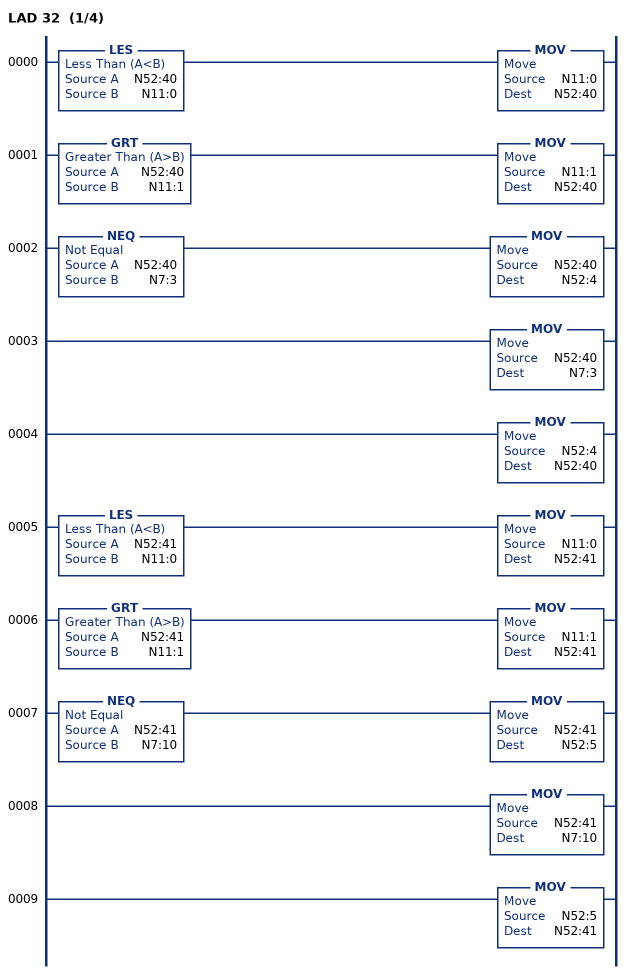
% Rung: 0 %
SOR LES N52:40 N11:0 MOV N11:0 N52:40 EOR
% Rung: 1 %
SOR GRT N52:40 N11:1 MOV N11:1 N52:40 EOR
% Rung: 2 %
SOR NEQ N52:40 N7:3 MOV N52:40 N52:4 EOR
% Rung: 3 %
SOR MOV N52:40 N7:3 EOR
% Rung: 4 %
SOR MOV N52:4 N52:40 EOR
% Rung: 5 %
SOR LES N52:41 N11:0 MOV N11:0 N52:41 EOR
% Rung: 6 %
SOR GRT N52:41 N11:1 MOV N11:1 N52:41 EOR
% Rung: 7 %
SOR NEQ N52:41 N7:10 MOV N52:41 N52:5 EOR
% Rung: 8 %
SOR MOV N52:41 N7:10 EOR
% Rung: 9 %
SOR MOV N52:5 N52:41 EOR

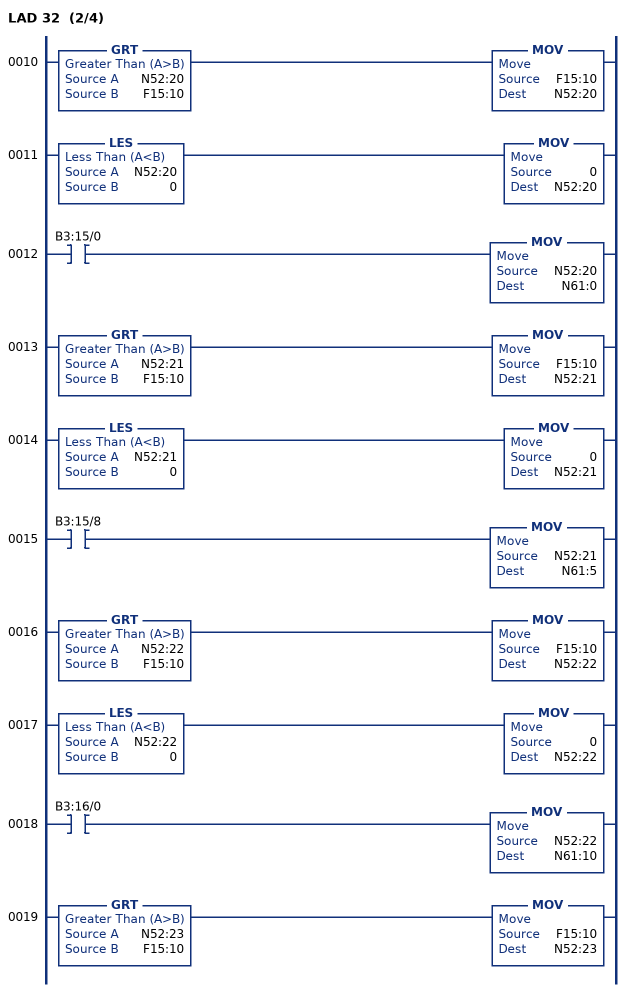
% Rung: 10 %
SOR GRT N52:20 F15:10 MOV F15:10 N52:20 EOR
% Rung: 11 %
SOR LES N52:20 0 MOV 0 N52:20 EOR
% Rung: 12 %
SOR XIC B3:15/0 MOV N52:20 N61:0 EOR
% Rung: 13 %
SOR GRT N52:21 F15:10 MOV F15:10 N52:21 EOR
% Rung: 14 %
SOR LES N52:21 0 MOV 0 N52:21 EOR
% Rung: 15 %
SOR XIC B3:15/8 MOV N52:21 N61:5 EOR
% Rung: 16 %
SOR GRT N52:22 F15:10 MOV F15:10 N52:22 EOR
% Rung: 17 %
SOR LES N52:22 0 MOV 0 N52:22 EOR
% Rung: 18 %
SOR XIC B3:16/0 MOV N52:22 N61:10 EOR
% Rung: 19 %
SOR GRT N52:23 F15:10 MOV F15:10 N52:23 EOR

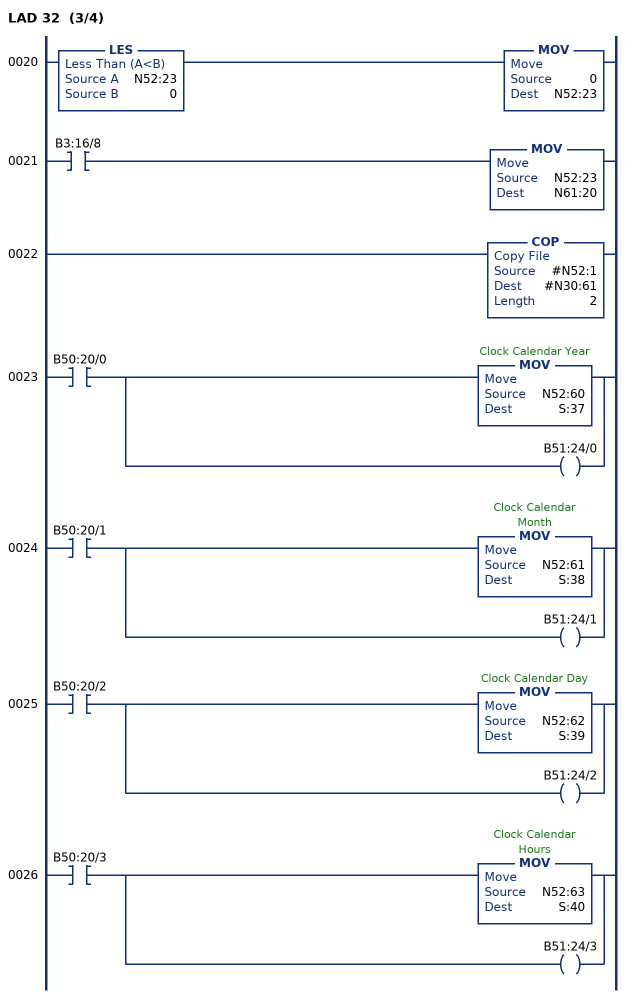
% Rung: 20 %
SOR LES N52:23 0 MOV 0 N52:23 EOR
% Rung: 21 %
SOR XIC B3:16/8 MOV N52:23 N61:20 EOR
% Rung: 22 %
SOR COP #N52:1 #N30:61 2 EOR
% Rung: 23 %
SOR XIC B50:20/0 BST MOV N52:60 S:37 NXB OTE B51:24/0 BND EOR
%   S:37  "Clock Calendar Year" %
% Rung: 24 %
SOR XIC B50:20/1 BST MOV N52:61 S:38 NXB OTE B51:24/1 BND EOR
%   S:38  "Clock Calendar Month" %
% Rung: 25 %
SOR XIC B50:20/2 BST MOV N52:62 S:39 NXB OTE B51:24/2 BND EOR
%   S:39  "Clock Calendar Day" %
% Rung: 26 %
SOR XIC B50:20/3 BST MOV N52:63 S:40 NXB OTE B51:24/3 BND EOR
%   S:40  "Clock Calendar Hours" %

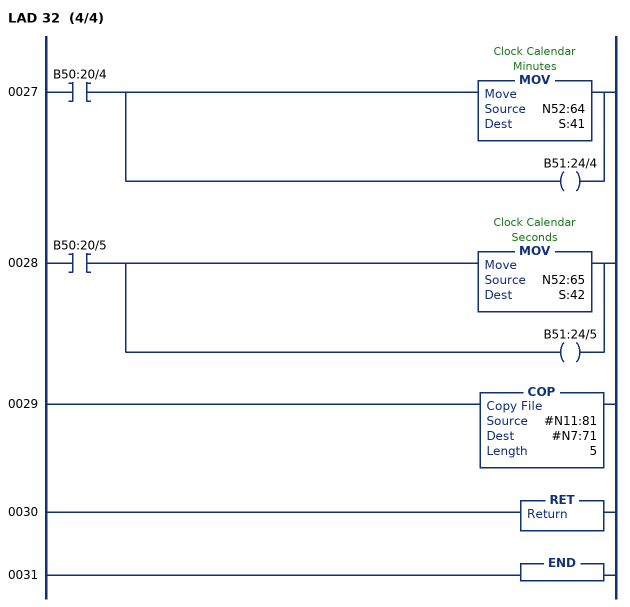
% Rung: 27 %
SOR XIC B50:20/4 BST MOV N52:64 S:41 NXB OTE B51:24/4 BND EOR
%   S:41  "Clock Calendar Minutes" %
% Rung: 28 %
SOR XIC B50:20/5 BST MOV N52:65 S:42 NXB OTE B51:24/5 BND EOR
%   S:42  "Clock Calendar Seconds" %
% Rung: 29 %
SOR COP #N11:81 #N7:71 5 EOR
% Rung: 30 %
SOR RET EOR
% Rung: 31 %
SOR END EOR

LADDER 33
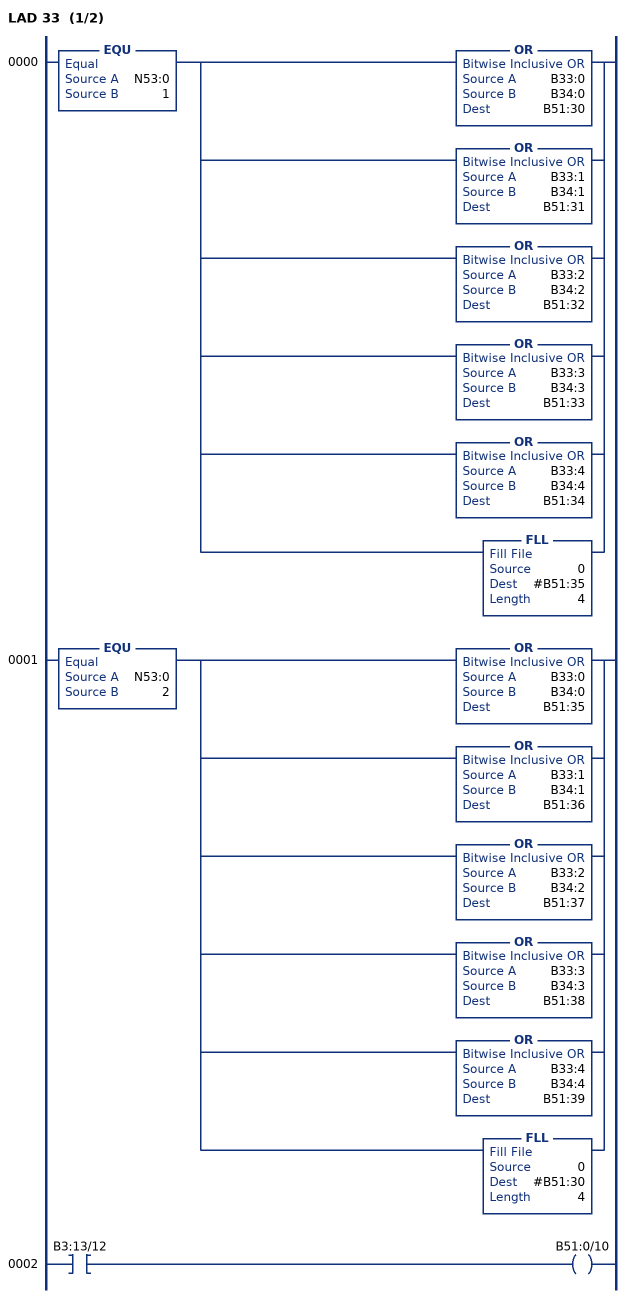
% Rung: 0 %
SOR EQU N53:0 1 BST OR B33:0 B34:0 B51:30 NXB OR B33:1 B34:1 B51:31 NXB OR B33:2 B34:2 B51:32 NXB OR B33:3 B34:3 B51:33 NXB OR B33:4 B34:4 B51:34 NXB FLL 0 #B51:35 4 BND EOR
% Rung: 1 %
SOR EQU N53:0 2 BST OR B33:0 B34:0 B51:35 NXB OR B33:1 B34:1 B51:36 NXB OR B33:2 B34:2 B51:37 NXB OR B33:3 B34:3 B51:38 NXB OR B33:4 B34:4 B51:39 NXB FLL 0 #B51:30 4 BND EOR
% Rung: 2 %
SOR XIC B3:13/12 OTE B51:0/10 EOR

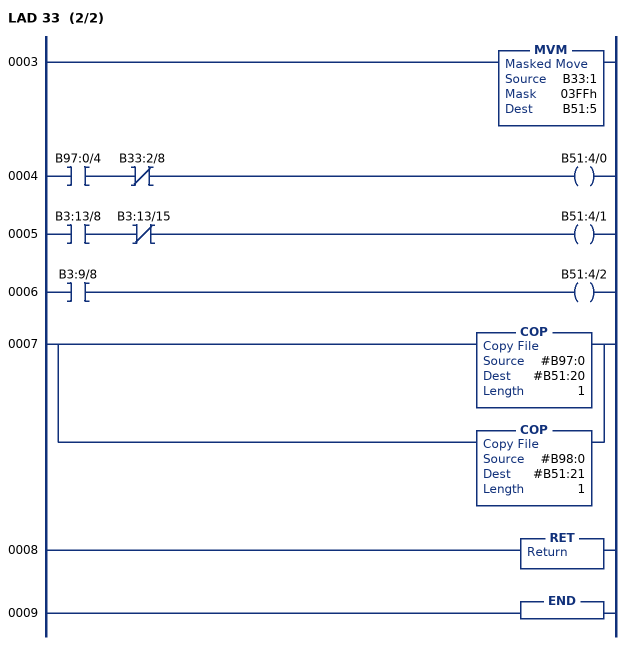
% Rung: 3 %
SOR MVM B33:1 03FFh B51:5 EOR
% Rung: 4 %
SOR XIC B97:0/4 XIO B33:2/8 OTE B51:4/0 EOR
% Rung: 5 %
SOR XIC B3:13/8 XIO B3:13/15 OTE B51:4/1 EOR
% Rung: 6 %
SOR XIC B3:9/8 OTE B51:4/2 EOR
% Rung: 7 %
SOR BST COP #B97:0 #B51:20 1 NXB COP #B98:0 #B51:21 1 BND EOR
% Rung: 8 %
SOR RET EOR
% Rung: 9 %
SOR END EOR

LADDER 34
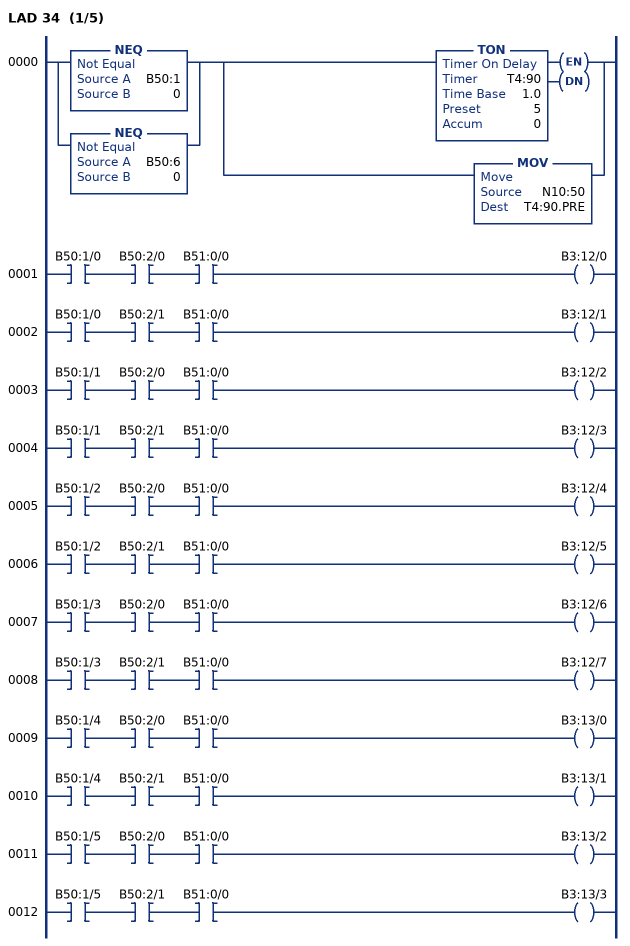
% Rung: 0 %
SOR BST NEQ B50:1 0 NXB NEQ B50:6 0 BND BST TON T4:90 1.0 5 0 NXB MOV N10:50 T4:90.PRE BND EOR
% Rung: 1 %
SOR XIC B50:1/0 XIC B50:2/0 XIC B51:0/0 OTE B3:12/0 EOR
% Rung: 2 %
SOR XIC B50:1/0 XIC B50:2/1 XIC B51:0/0 OTE B3:12/1 EOR
% Rung: 3 %
SOR XIC B50:1/1 XIC B50:2/0 XIC B51:0/0 OTE B3:12/2 EOR
% Rung: 4 %
SOR XIC B50:1/1 XIC B50:2/1 XIC B51:0/0 OTE B3:12/3 EOR
% Rung: 5 %
SOR XIC B50:1/2 XIC B50:2/0 XIC B51:0/0 OTE B3:12/4 EOR
% Rung: 6 %
SOR XIC B50:1/2 XIC B50:2/1 XIC B51:0/0 OTE B3:12/5 EOR
% Rung: 7 %
SOR XIC B50:1/3 XIC B50:2/0 XIC B51:0/0 OTE B3:12/6 EOR
% Rung: 8 %
SOR XIC B50:1/3 XIC B50:2/1 XIC B51:0/0 OTE B3:12/7 EOR
% Rung: 9 %
SOR XIC B50:1/4 XIC B50:2/0 XIC B51:0/0 OTE B3:13/0 EOR
% Rung: 10 %
SOR XIC B50:1/4 XIC B50:2/1 XIC B51:0/0 OTE B3:13/1 EOR
% Rung: 11 %
SOR XIC B50:1/5 XIC B50:2/0 XIC B51:0/0 OTE B3:13/2 EOR
% Rung: 12 %
SOR XIC B50:1/5 XIC B50:2/1 XIC B51:0/0 OTE B3:13/3 EOR

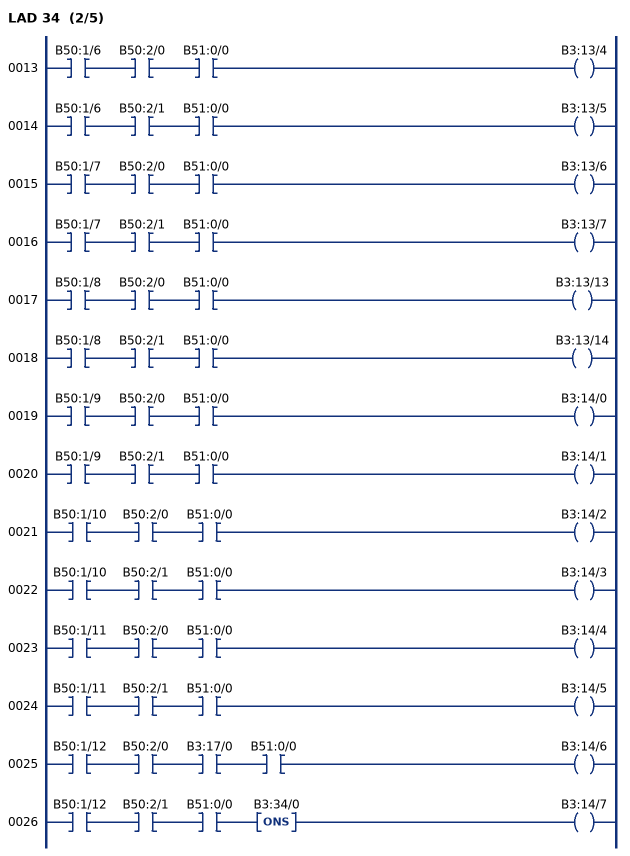
% Rung: 13 %
SOR XIC B50:1/6 XIC B50:2/0 XIC B51:0/0 OTE B3:13/4 EOR
% Rung: 14 %
SOR XIC B50:1/6 XIC B50:2/1 XIC B51:0/0 OTE B3:13/5 EOR
% Rung: 15 %
SOR XIC B50:1/7 XIC B50:2/0 XIC B51:0/0 OTE B3:13/6 EOR
% Rung: 16 %
SOR XIC B50:1/7 XIC B50:2/1 XIC B51:0/0 OTE B3:13/7 EOR
% Rung: 17 %
SOR XIC B50:1/8 XIC B50:2/0 XIC B51:0/0 OTE B3:13/13 EOR
% Rung: 18 %
SOR XIC B50:1/8 XIC B50:2/1 XIC B51:0/0 OTE B3:13/14 EOR
% Rung: 19 %
SOR XIC B50:1/9 XIC B50:2/0 XIC B51:0/0 OTE B3:14/0 EOR
% Rung: 20 %
SOR XIC B50:1/9 XIC B50:2/1 XIC B51:0/0 OTE B3:14/1 EOR
% Rung: 21 %
SOR XIC B50:1/10 XIC B50:2/0 XIC B51:0/0 OTE B3:14/2 EOR
% Rung: 22 %
SOR XIC B50:1/10 XIC B50:2/1 XIC B51:0/0 OTE B3:14/3 EOR
% Rung: 23 %
SOR XIC B50:1/11 XIC B50:2/0 XIC B51:0/0 OTE B3:14/4 EOR
% Rung: 24 %
SOR XIC B50:1/11 XIC B50:2/1 XIC B51:0/0 OTE B3:14/5 EOR
% Rung: 25 %
SOR XIC B50:1/12 XIC B50:2/0 XIC B3:17/0 XIC B51:0/0 OTE B3:14/6 EOR
% Rung: 26 %
SOR XIC B50:1/12 XIC B50:2/1 XIC B51:0/0 OSR B3:34/0 OTE B3:14/7 EOR

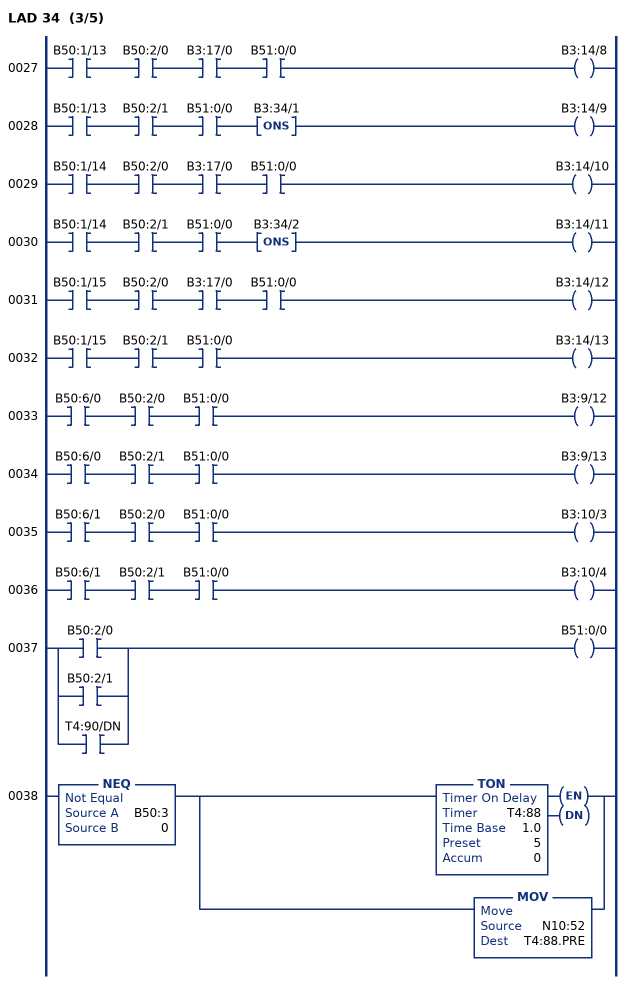
% Rung: 27 %
SOR XIC B50:1/13 XIC B50:2/0 XIC B3:17/0 XIC B51:0/0 OTE B3:14/8 EOR
% Rung: 28 %
SOR XIC B50:1/13 XIC B50:2/1 XIC B51:0/0 OSR B3:34/1 OTE B3:14/9 EOR
% Rung: 29 %
SOR XIC B50:1/14 XIC B50:2/0 XIC B3:17/0 XIC B51:0/0 OTE B3:14/10 EOR
% Rung: 30 %
SOR XIC B50:1/14 XIC B50:2/1 XIC B51:0/0 OSR B3:34/2 OTE B3:14/11 EOR
% Rung: 31 %
SOR XIC B50:1/15 XIC B50:2/0 XIC B3:17/0 XIC B51:0/0 OTE B3:14/12 EOR
% Rung: 32 %
SOR XIC B50:1/15 XIC B50:2/1 XIC B51:0/0 OTE B3:14/13 EOR
% Rung: 33 %
SOR XIC B50:6/0 XIC B50:2/0 XIC B51:0/0 OTE B3:9/12 EOR
% Rung: 34 %
SOR XIC B50:6/0 XIC B50:2/1 XIC B51:0/0 OTE B3:9/13 EOR
% Rung: 35 %
SOR XIC B50:6/1 XIC B50:2/0 XIC B51:0/0 OTE B3:10/3 EOR
% Rung: 36 %
SOR XIC B50:6/1 XIC B50:2/1 XIC B51:0/0 OTE B3:10/4 EOR
% Rung: 37 %
SOR BST XIC B50:2/0 NXB XIC B50:2/1 NXB XIC T4:90/DN BND OTE B51:0/0 EOR
% Rung: 38 %
SOR NEQ B50:3 0 BST TON T4:88 1.0 5 0 NXB MOV N10:52 T4:88.PRE BND EOR

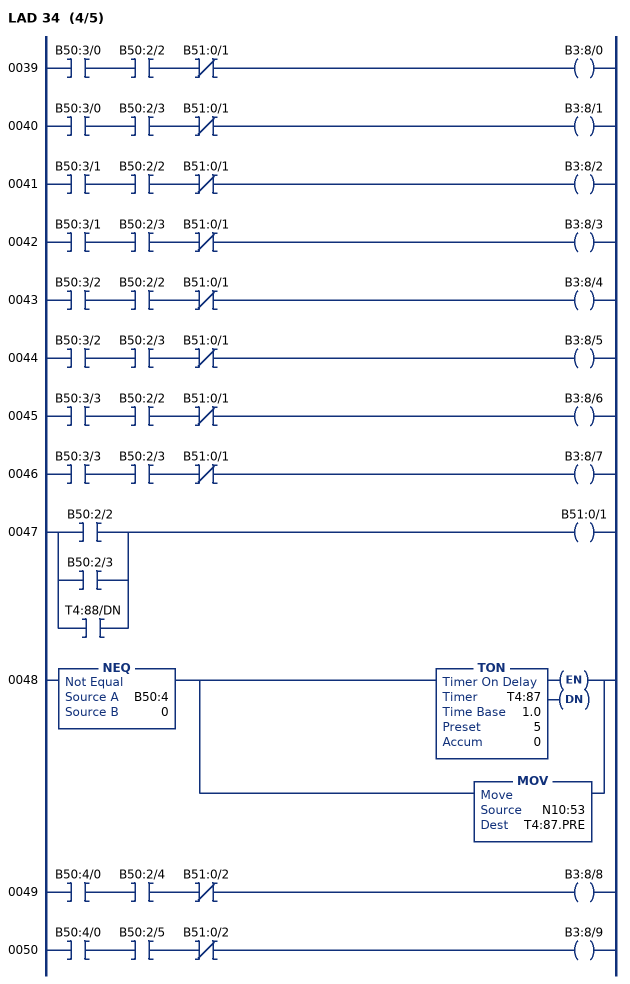
% Rung: 39 %
SOR XIC B50:3/0 XIC B50:2/2 XIO B51:0/1 OTE B3:8/0 EOR
% Rung: 40 %
SOR XIC B50:3/0 XIC B50:2/3 XIO B51:0/1 OTE B3:8/1 EOR
% Rung: 41 %
SOR XIC B50:3/1 XIC B50:2/2 XIO B51:0/1 OTE B3:8/2 EOR
% Rung: 42 %
SOR XIC B50:3/1 XIC B50:2/3 XIO B51:0/1 OTE B3:8/3 EOR
% Rung: 43 %
SOR XIC B50:3/2 XIC B50:2/2 XIO B51:0/1 OTE B3:8/4 EOR
% Rung: 44 %
SOR XIC B50:3/2 XIC B50:2/3 XIO B51:0/1 OTE B3:8/5 EOR
% Rung: 45 %
SOR XIC B50:3/3 XIC B50:2/2 XIO B51:0/1 OTE B3:8/6 EOR
% Rung: 46 %
SOR XIC B50:3/3 XIC B50:2/3 XIO B51:0/1 OTE B3:8/7 EOR
% Rung: 47 %
SOR BST XIC B50:2/2 NXB XIC B50:2/3 NXB XIC T4:88/DN BND OTE B51:0/1 EOR
% Rung: 48 %
SOR NEQ B50:4 0 BST TON T4:87 1.0 5 0 NXB MOV N10:53 T4:87.PRE BND EOR
% Rung: 49 %
SOR XIC B50:4/0 XIC B50:2/4 XIO B51:0/2 OTE B3:8/8 EOR
% Rung: 50 %
SOR XIC B50:4/0 XIC B50:2/5 XIO B51:0/2 OTE B3:8/9 EOR

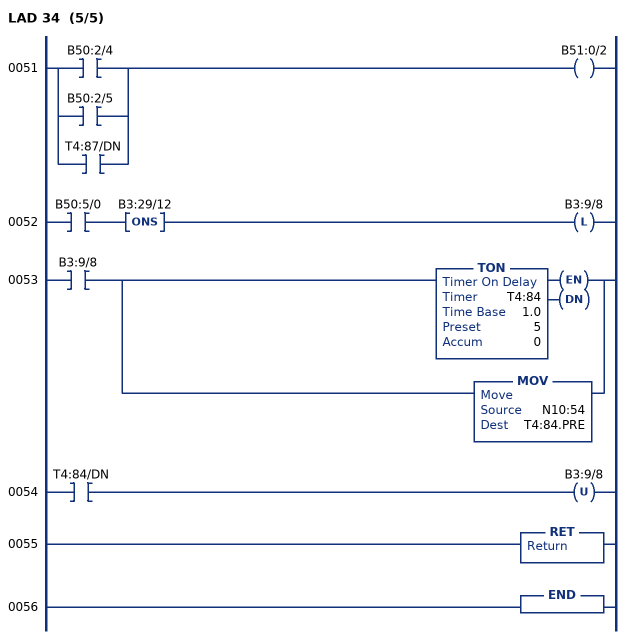
% Rung: 51 %
SOR BST XIC B50:2/4 NXB XIC B50:2/5 NXB XIC T4:87/DN BND OTE B51:0/2 EOR
% Rung: 52 %
SOR XIC B50:5/0 OSR B3:29/12 OTL B3:9/8 EOR
% Rung: 53 %
SOR XIC B3:9/8 BST TON T4:84 1.0 5 0 NXB MOV N10:54 T4:84.PRE BND EOR
% Rung: 54 %
SOR XIC T4:84/DN OTU B3:9/8 EOR
% Rung: 55 %
SOR RET EOR
% Rung: 56 %
SOR END EOR

LADDER 35
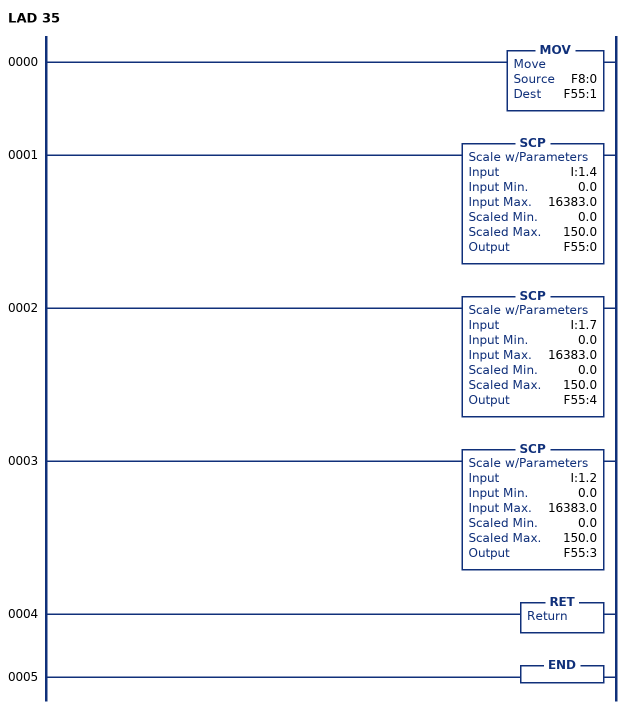
% Rung: 0 %
SOR MOV F8:0 F55:1 EOR
% Rung: 1 %
SOR SCP I:1.4 0.0 16383.0 0.0 150.0 F55:0 EOR
% Rung: 2 %
SOR SCP I:1.7 0.0 16383.0 0.0 150.0 F55:4 EOR
% Rung: 3 %
SOR SCP I:1.2 0.0 16383.0 0.0 150.0 F55:3 EOR
% Rung: 4 %
SOR RET EOR
% Rung: 5 %
SOR END EOR

LADDER 36
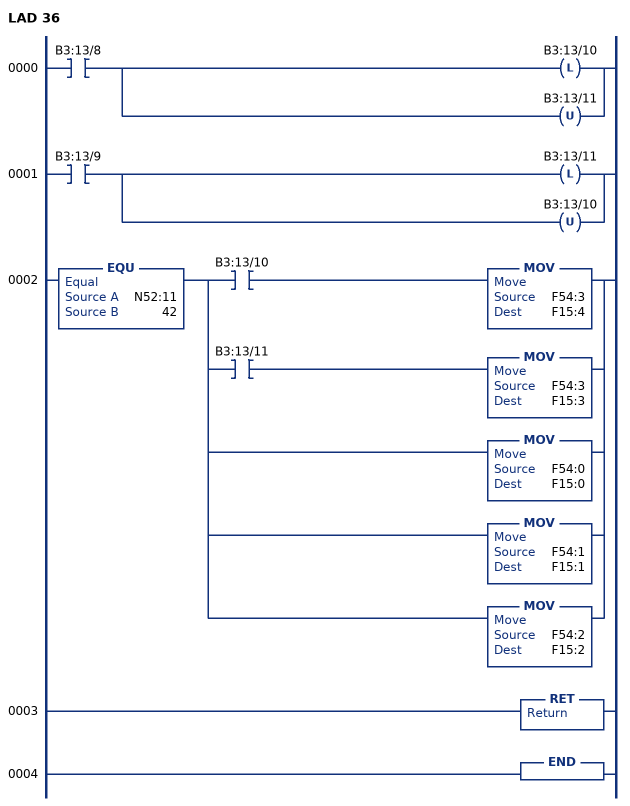
% Rung: 0 %
SOR XIC B3:13/8 BST OTL B3:13/10 NXB OTU B3:13/11 BND EOR
% Rung: 1 %
SOR XIC B3:13/9 BST OTL B3:13/11 NXB OTU B3:13/10 BND EOR
% Rung: 2 %
SOR EQU N52:11 42 BST XIC B3:13/10 MOV F54:3 F15:4 NXB XIC B3:13/11 MOV F54:3 F15:3 NXB MOV F54:0 F15:0 NXB MOV F54:1 F15:1 NXB MOV F54:2 F15:2 BND EOR
% Rung: 3 %
SOR RET EOR
% Rung: 4 %
SOR END EOR

LADDER 37
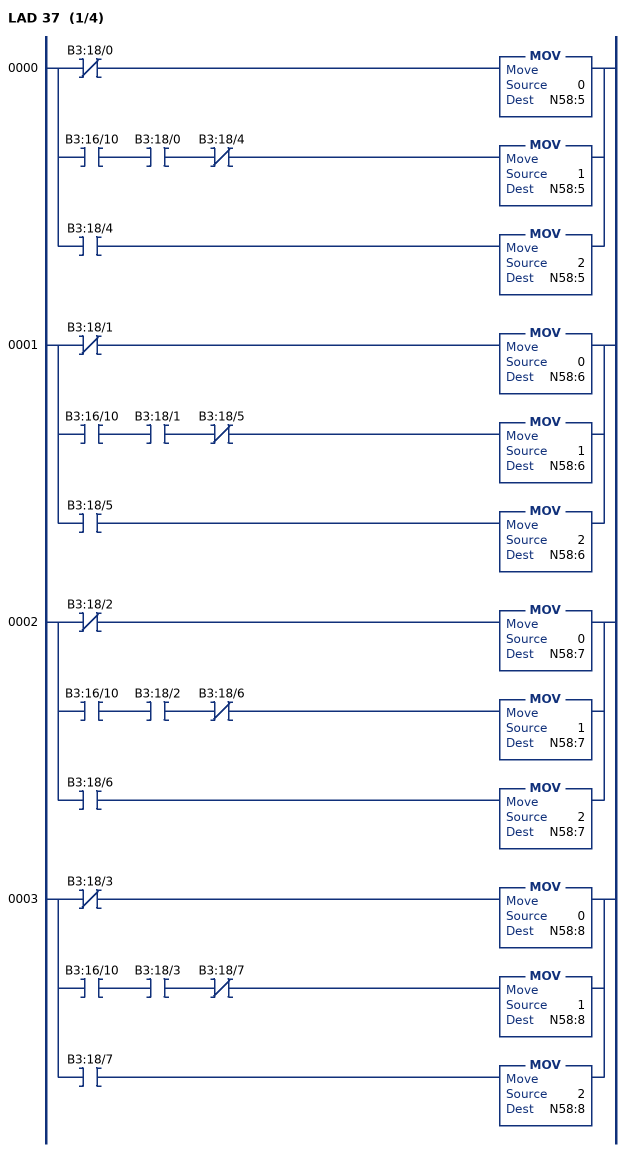
% Rung: 0 %
SOR BST XIO B3:18/0 MOV 0 N58:5 NXB XIC B3:16/10 XIC B3:18/0 XIO B3:18/4 MOV 1 N58:5 NXB XIC B3:18/4 MOV 2 N58:5 BND EOR
% Rung: 1 %
SOR BST XIO B3:18/1 MOV 0 N58:6 NXB XIC B3:16/10 XIC B3:18/1 XIO B3:18/5 MOV 1 N58:6 NXB XIC B3:18/5 MOV 2 N58:6 BND EOR
% Rung: 2 %
SOR BST XIO B3:18/2 MOV 0 N58:7 NXB XIC B3:16/10 XIC B3:18/2 XIO B3:18/6 MOV 1 N58:7 NXB XIC B3:18/6 MOV 2 N58:7 BND EOR
% Rung: 3 %
SOR BST XIO B3:18/3 MOV 0 N58:8 NXB XIC B3:16/10 XIC B3:18/3 XIO B3:18/7 MOV 1 N58:8 NXB XIC B3:18/7 MOV 2 N58:8 BND EOR

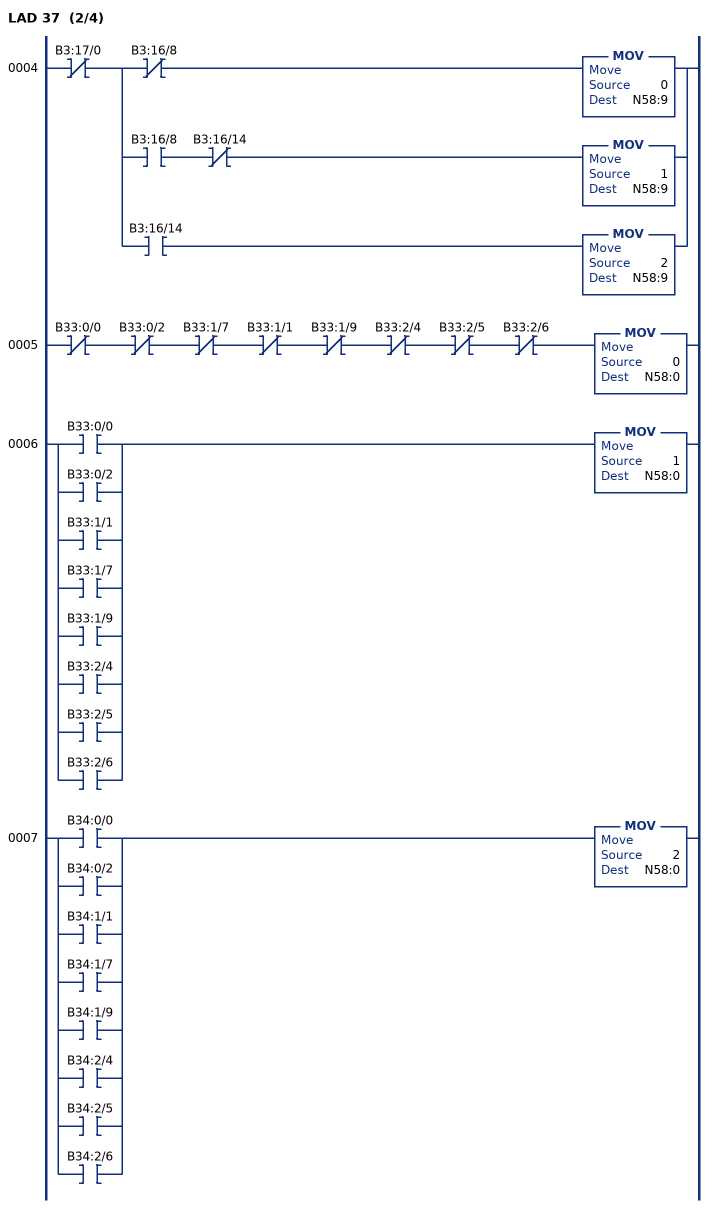
% Rung: 4 %
SOR XIO B3:17/0 BST XIO B3:16/8 MOV 0 N58:9 NXB XIC B3:16/8 XIO B3:16/14 MOV 1 N58:9 NXB XIC B3:16/14 MOV 2 N58:9 BND EOR
% Rung: 5 %
SOR XIO B33:0/0 XIO B33:0/2 XIO B33:1/7 XIO B33:1/1 XIO B33:1/9 XIO B33:2/4 XIO B33:2/5 XIO B33:2/6 MOV 0 N58:0 EOR
% Rung: 6 %
SOR BST XIC B33:0/0 NXB XIC B33:0/2 NXB XIC B33:1/1 NXB XIC B33:1/7 NXB XIC B33:1/9 NXB XIC B33:2/4 NXB XIC B33:2/5 NXB XIC B33:2/6 BND MOV 1 N58:0 EOR
% Rung: 7 %
SOR BST XIC B34:0/0 NXB XIC B34:0/2 NXB XIC B34:1/1 NXB XIC B34:1/7 NXB XIC B34:1/9 NXB XIC B34:2/4 NXB XIC B34:2/5 NXB XIC B34:2/6 BND MOV 2 N58:0 EOR

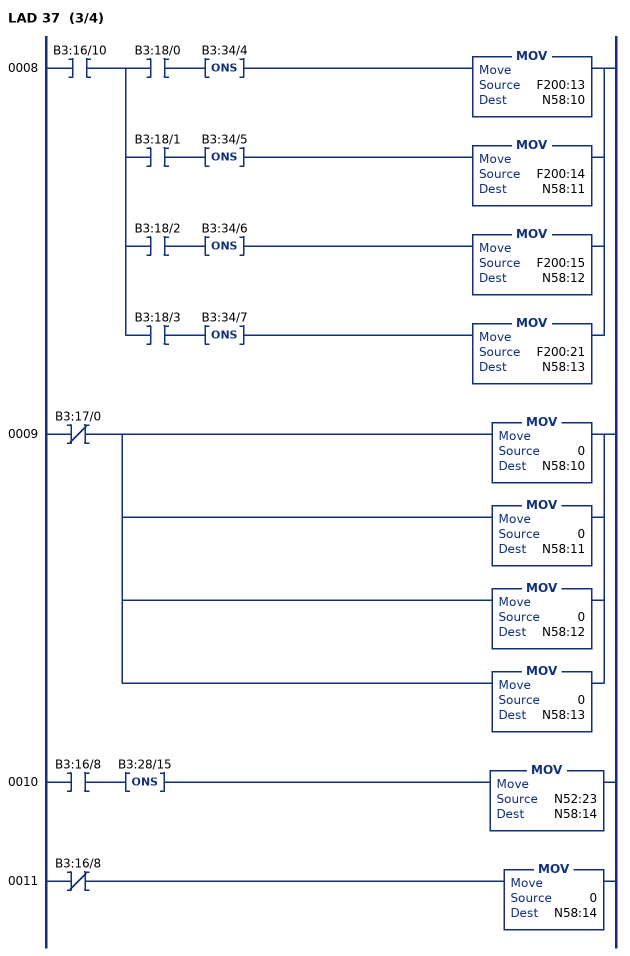
% Rung: 8 %
SOR XIC B3:16/10 BST XIC B3:18/0 OSR B3:34/4 MOV F200:13 N58:10 NXB XIC B3:18/1 OSR B3:34/5 MOV F200:14 N58:11 NXB XIC B3:18/2 OSR B3:34/6 MOV F200:15 N58:12 NXB XIC B3:18/3 OSR B3:34/7 MOV F200:21 N58:13 BND EOR
% Rung: 9 %
SOR XIO B3:17/0 BST MOV 0 N58:10 NXB MOV 0 N58:11 NXB MOV 0 N58:12 NXB MOV 0 N58:13 BND EOR
% Rung: 10 %
SOR XIC B3:16/8 OSR B3:28/15 MOV N52:23 N58:14 EOR
% Rung: 11 %
SOR XIO B3:16/8 MOV 0 N58:14 EOR

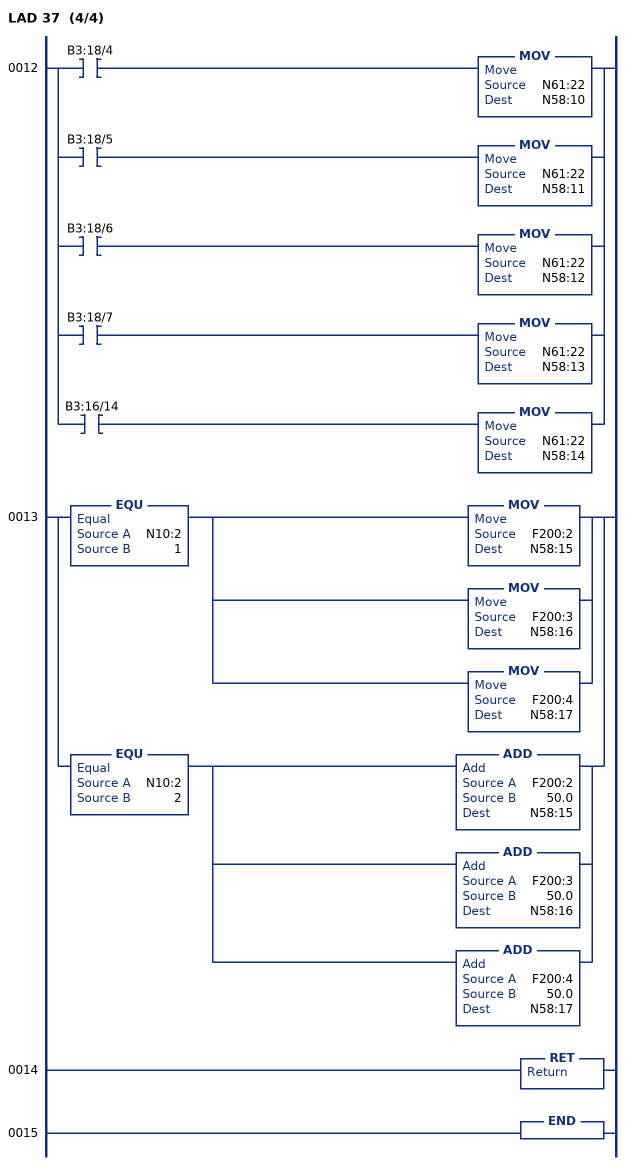
% Rung: 12 %
SOR BST XIC B3:18/4 MOV N61:22 N58:10 NXB XIC B3:18/5 MOV N61:22 N58:11 NXB XIC B3:18/6 MOV N61:22 N58:12 NXB XIC B3:18/7 MOV N61:22 N58:13 NXB XIC B3:16/14 MOV N61:22 N58:14 BND EOR
% Rung: 13 %
SOR BST EQU N10:2 1 BST MOV F200:2 N58:15 NXB MOV F200:3 N58:16 NXB MOV F200:4 N58:17 BND NXB EQU N10:2 2 BST ADD F200:2 50.0 N58:15 NXB ADD F200:3 50.0 N58:16 NXB ADD F200:4 50.0 N58:17 BND BND EOR
% Rung: 14 %
SOR RET EOR
% Rung: 15 %
SOR END EOR

LADDER 38
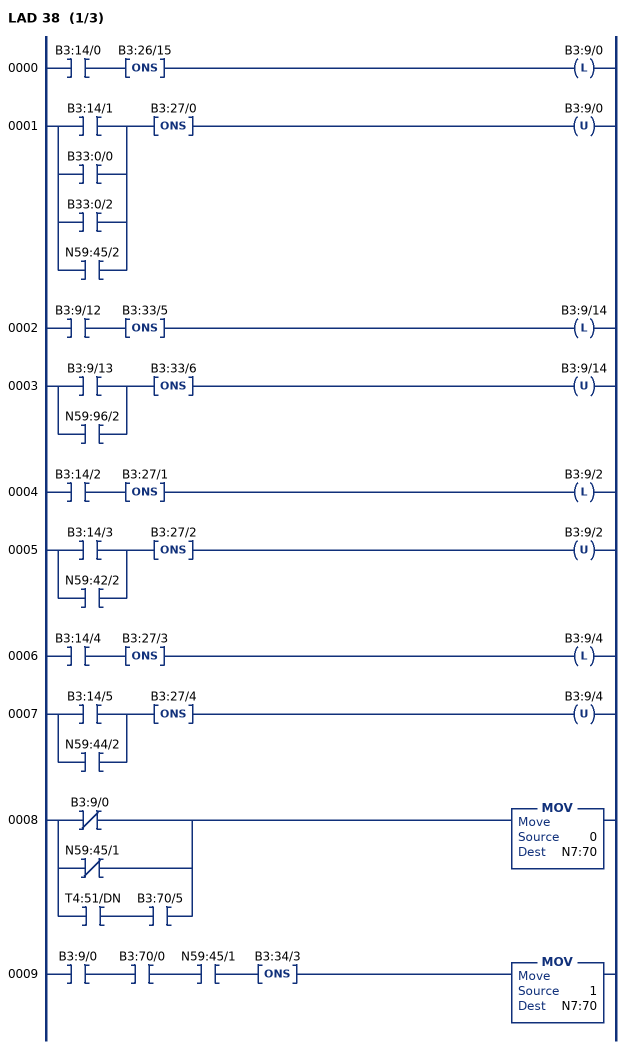
% Rung: 0 %
SOR XIC B3:14/0 OSR B3:26/15 OTL B3:9/0 EOR
% Rung: 1 %
SOR BST XIC B3:14/1 NXB XIC B33:0/0 NXB XIC B33:0/2 NXB XIC N59:45/2 BND OSR B3:27/0 OTU B3:9/0 EOR
% Rung: 2 %
SOR XIC B3:9/12 OSR B3:33/5 OTL B3:9/14 EOR
% Rung: 3 %
SOR BST XIC B3:9/13 NXB XIC N59:96/2 BND OSR B3:33/6 OTU B3:9/14 EOR
% Rung: 4 %
SOR XIC B3:14/2 OSR B3:27/1 OTL B3:9/2 EOR
% Rung: 5 %
SOR BST XIC B3:14/3 NXB XIC N59:42/2 BND OSR B3:27/2 OTU B3:9/2 EOR
% Rung: 6 %
SOR XIC B3:14/4 OSR B3:27/3 OTL B3:9/4 EOR
% Rung: 7 %
SOR BST XIC B3:14/5 NXB XIC N59:44/2 BND OSR B3:27/4 OTU B3:9/4 EOR
% Rung: 8 %
SOR BST XIO B3:9/0 NXB XIO N59:45/1 NXB XIC T4:51/DN XIC B3:70/5 BND MOV 0 N7:70 EOR
% Rung: 9 %
SOR XIC B3:9/0 XIC B3:70/0 XIC N59:45/1 OSR B3:34/3 MOV 1 N7:70 EOR

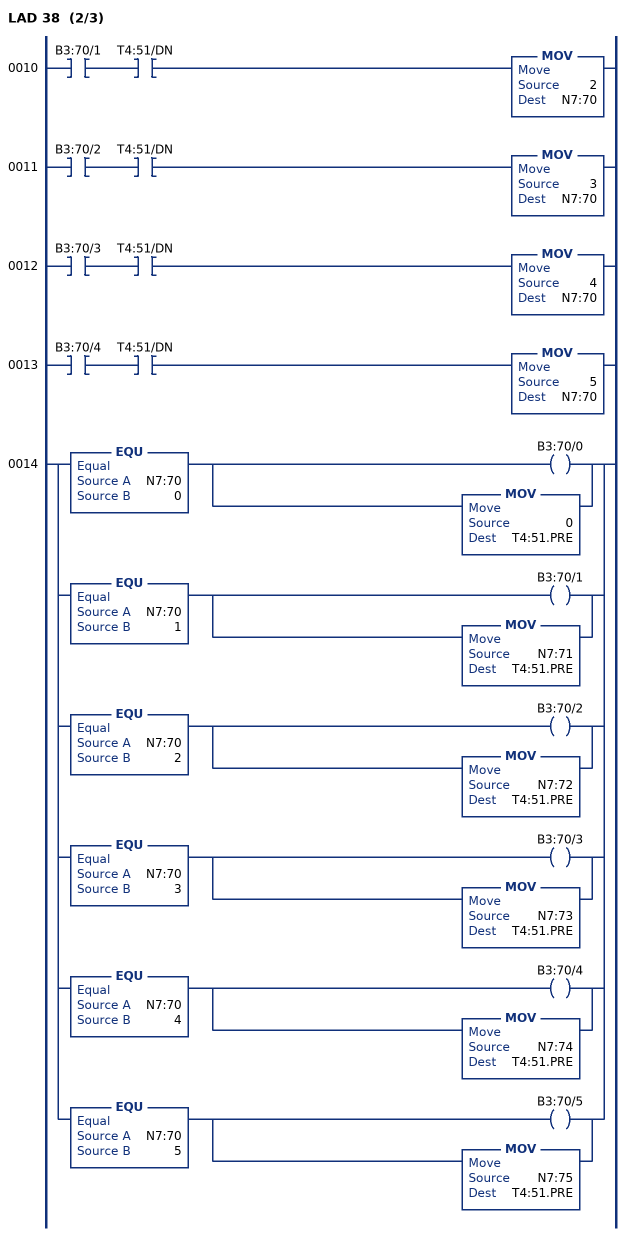
% Rung: 10 %
SOR XIC B3:70/1 XIC T4:51/DN MOV 2 N7:70 EOR
% Rung: 11 %
SOR XIC B3:70/2 XIC T4:51/DN MOV 3 N7:70 EOR
% Rung: 12 %
SOR XIC B3:70/3 XIC T4:51/DN MOV 4 N7:70 EOR
% Rung: 13 %
SOR XIC B3:70/4 XIC T4:51/DN MOV 5 N7:70 EOR
% Rung: 14 %
SOR BST EQU N7:70 0 BST OTE B3:70/0 NXB MOV 0 T4:51.PRE BND NXB EQU N7:70 1 BST OTE B3:70/1 NXB MOV N7:71 T4:51.PRE BND NXB EQU N7:70 2 BST OTE B3:70/2 NXB MOV N7:72 T4:51.PRE BND NXB EQU N7:70 3 BST OTE B3:70/3 NXB MOV N7:73 T4:51.PRE BND NXB EQU N7:70 4 BST OTE B3:70/4 NXB MOV N7:74 T4:51.PRE BND NXB EQU N7:70 5 BST OTE B3:70/5 NXB MOV N7:75 T4:51.PRE BND BND EOR

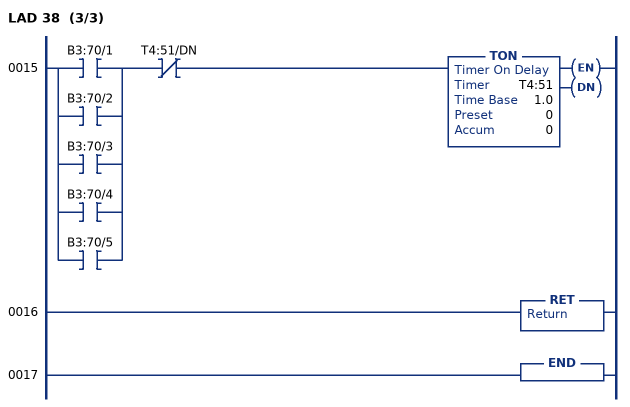
% Rung: 15 %
SOR BST XIC B3:70/1 NXB XIC B3:70/2 NXB XIC B3:70/3 NXB XIC B3:70/4 NXB XIC B3:70/5 BND XIO T4:51/DN TON T4:51 1.0 0 0 EOR
% Rung: 16 %
SOR RET EOR
% Rung: 17 %
SOR END EOR

LADDER 39
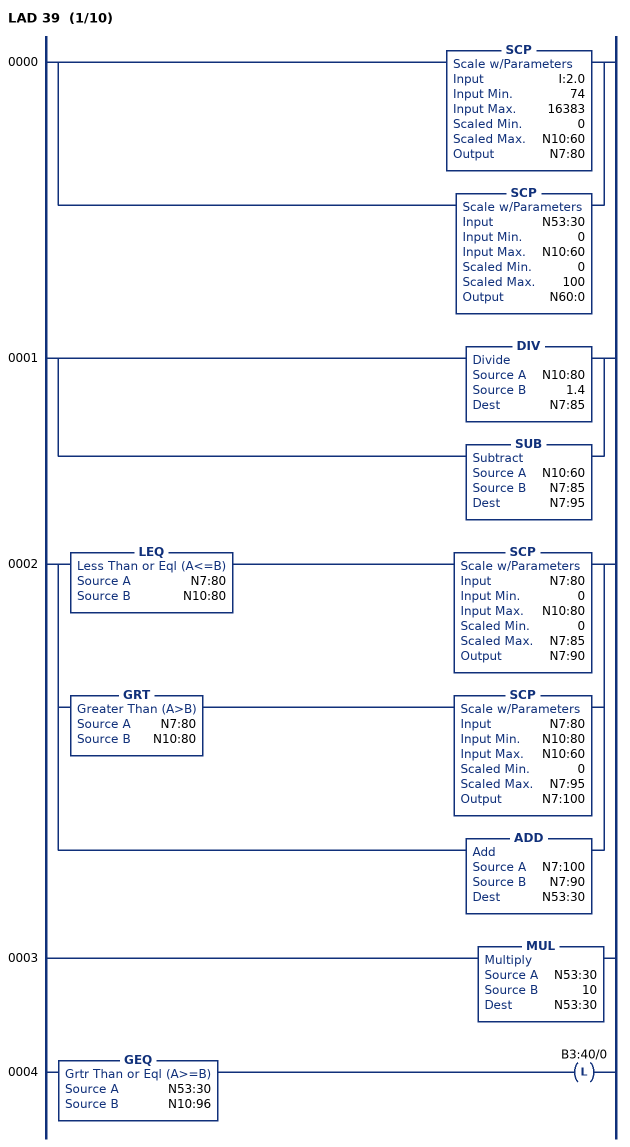
% Rung: 0 %
SOR BST SCP I:2.0 74 16383 0 N10:60 N7:80 NXB SCP N53:30 0 N10:60 0 100 N60:0 BND EOR
% Rung: 1 %
SOR BST DIV N10:80 1.4 N7:85 NXB SUB N10:60 N7:85 N7:95 BND EOR
% Rung: 2 %
SOR BST LEQ N7:80 N10:80 SCP N7:80 0 N10:80 0 N7:85 N7:90 NXB GRT N7:80 N10:80 SCP N7:80 N10:80 N10:60 0 N7:95 N7:100 NXB ADD N7:100 N7:90 N53:30 BND EOR
% Rung: 3 %
SOR MUL N53:30 10 N53:30 EOR
% Rung: 4 %
SOR GEQ N53:30 N10:96 OTL B3:40/0 EOR

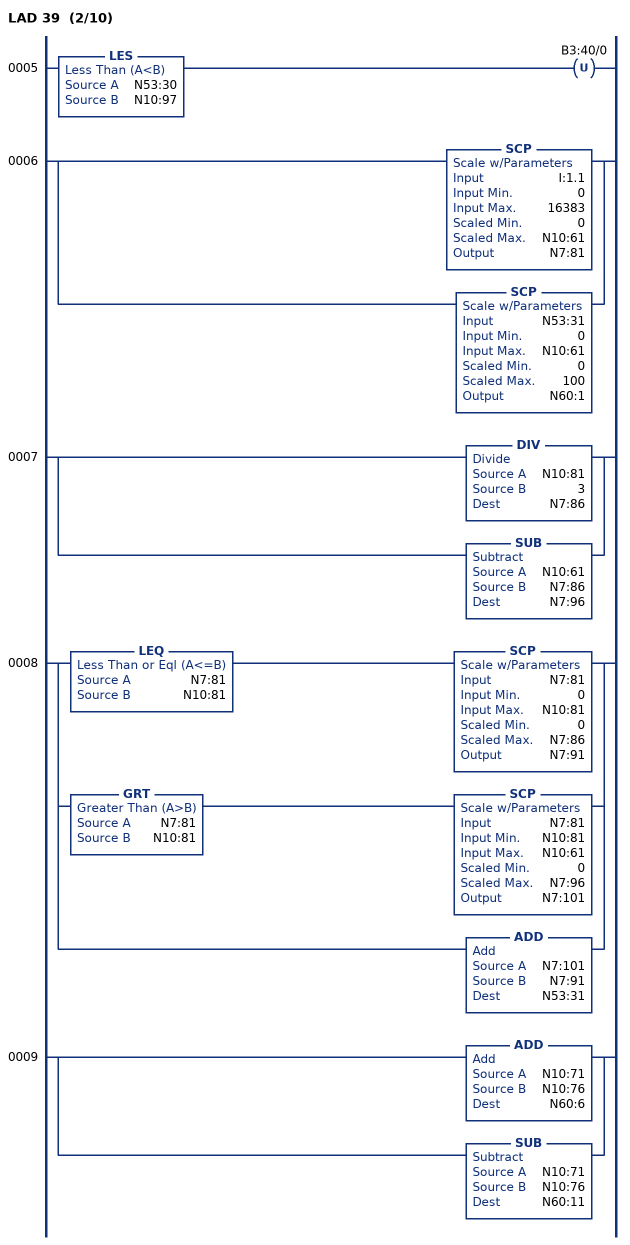
% Rung: 5 %
SOR LES N53:30 N10:97 OTU B3:40/0 EOR
% Rung: 6 %
SOR BST SCP I:1.1 0 16383 0 N10:61 N7:81 NXB SCP N53:31 0 N10:61 0 100 N60:1 BND EOR
% Rung: 7 %
SOR BST DIV N10:81 3 N7:86 NXB SUB N10:61 N7:86 N7:96 BND EOR
% Rung: 8 %
SOR BST LEQ N7:81 N10:81 SCP N7:81 0 N10:81 0 N7:86 N7:91 NXB GRT N7:81 N10:81 SCP N7:81 N10:81 N10:61 0 N7:96 N7:101 NXB ADD N7:101 N7:91 N53:31 BND EOR
% Rung: 9 %
SOR BST ADD N10:71 N10:76 N60:6 NXB SUB N10:71 N10:76 N60:11 BND EOR

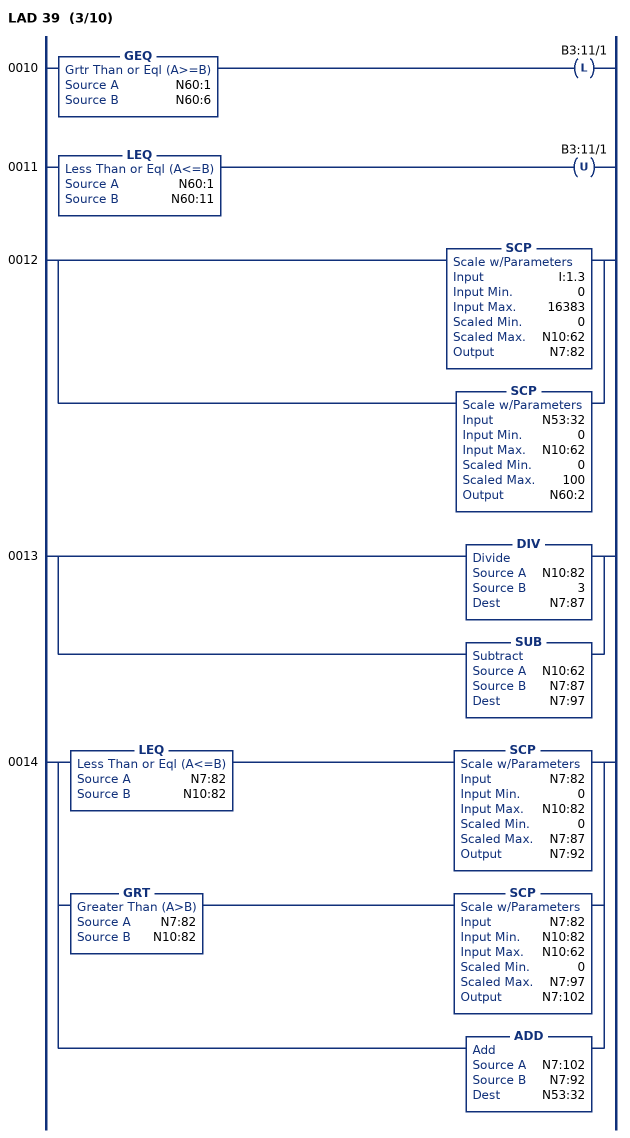
% Rung: 10 %
SOR GEQ N60:1 N60:6 OTL B3:11/1 EOR
% Rung: 11 %
SOR LEQ N60:1 N60:11 OTU B3:11/1 EOR
% Rung: 12 %
SOR BST SCP I:1.3 0 16383 0 N10:62 N7:82 NXB SCP N53:32 0 N10:62 0 100 N60:2 BND EOR
% Rung: 13 %
SOR BST DIV N10:82 3 N7:87 NXB SUB N10:62 N7:87 N7:97 BND EOR
% Rung: 14 %
SOR BST LEQ N7:82 N10:82 SCP N7:82 0 N10:82 0 N7:87 N7:92 NXB GRT N7:82 N10:82 SCP N7:82 N10:82 N10:62 0 N7:97 N7:102 NXB ADD N7:102 N7:92 N53:32 BND EOR

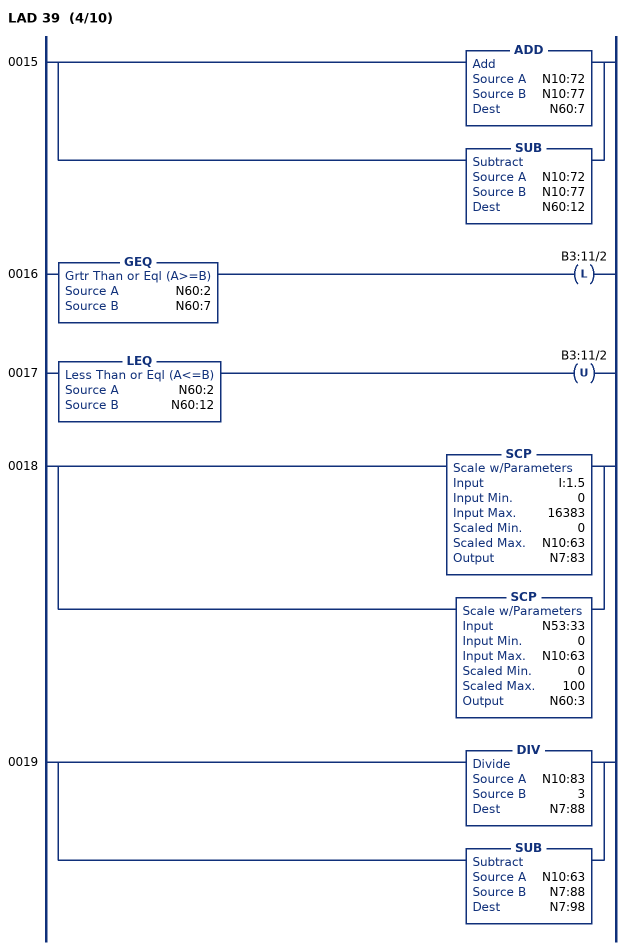
% Rung: 15 %
SOR BST ADD N10:72 N10:77 N60:7 NXB SUB N10:72 N10:77 N60:12 BND EOR
% Rung: 16 %
SOR GEQ N60:2 N60:7 OTL B3:11/2 EOR
% Rung: 17 %
SOR LEQ N60:2 N60:12 OTU B3:11/2 EOR
% Rung: 18 %
SOR BST SCP I:1.5 0 16383 0 N10:63 N7:83 NXB SCP N53:33 0 N10:63 0 100 N60:3 BND EOR
% Rung: 19 %
SOR BST DIV N10:83 3 N7:88 NXB SUB N10:63 N7:88 N7:98 BND EOR

